FUNCTION_BLOCK FB_Snake EXTENDS FB_Glowny
VAR

	poleGry:S_Macierz;	
	
	wiersz:INT;//potem usunąć oba
	kolumna:INT;
	
	stanGry:INT:=3;

	iLicznikPrendkosci: INT;

	
	GAMEOVER:BOOL:=TRUE;
	EKRANSTARTOWY:BOOL:=FALSE;
	
	kierunek: INT;
	iLicznikKierunku: INT;
	kierunekRuchu:E_kierunek;
	
	stanJedzenia:BOOL;
	jedzeniePozycjaX:INT;
	jedzeniePozycjaY:INT;
	
	iLicnikPunktow:INT:=1;
	
	iWektorOgonaX:ARRAY[2..400] OF INT;
	iWektorOgonaY:ARRAY[2..400] OF INT;
	iLicznikY:INT:=2;

END_VAR

CASE stanGry OF
	
0:	
	FOR iLicznikKierunku:=1 TO 4  DO
		IF GVL_Lista.bStanStrzalek[iLicznikKierunku]=TRUE THEN
			kierunek:=iLicznikKierunku;							//sprawdzanie obecnego kierunku ruchu
			IF kierunek=1 THEN
				kierunekRuchu:=1;
			END_IF
			IF kierunek=2 THEN
				kierunekRuchu:=2;
			END_IF
			IF kierunek=3 THEN
				kierunekRuchu:=3;
			END_IF
			IF kierunek=4 THEN
				kierunekRuchu:=4;
			END_IF
		END_IF
	END_FOR
	M_SprawdzanieKolizji();
	IF stanJedzenia=FALSE THEN									//jeśli zdobędziemy punkt generuje nowe do zdobycia
		M_GenerowanieJedzenia();
	END_IF
	
	SUPER^.timerRuchu(IN:=TRUE,PT:=INT_TO_TIME(1000-(iLicznikPrendkosci*iLicnikPunktow))); //czas pomiędzy kolejnymi rychami 
	IF timerRuchu.Q=TRUE THEN
		IF  kierunek=1 THEN						//lewo
			iLicznikY:=iLicznikY+1;
			iWektorOgonaX[iLicznikY]:=wiersz;
			iWektorOgonaY[iLicznikY]:=kolumna;
			wiersz:=wiersz-1;
		END_IF
		
		IF  kierunek=2 THEN						//dół
			iLicznikY:=iLicznikY+1;
			iWektorOgonaX[iLicznikY]:=wiersz;
			iWektorOgonaY[iLicznikY]:=kolumna;
			kolumna:=kolumna+1;
			
		END_IF
		
		IF  kierunek=3 THEN						//prawo
			iLicznikY:=iLicznikY+1;
			iWektorOgonaX[iLicznikY]:=wiersz;
			iWektorOgonaY[iLicznikY]:=kolumna;
			wiersz:=wiersz+1;
			
		END_IF
		
		IF  kierunek=4 THEN						//góra
			iLicznikY:=iLicznikY+1;
			iWektorOgonaX[iLicznikY]:=wiersz;
			iWektorOgonaY[iLicznikY]:=kolumna;
			kolumna:=kolumna-1;
			
		END_IF
		
		stanGry:=1;
		
		IF kolumna>10 OR wiersz>10 OR kolumna<1 OR wiersz<1 THEN	// detekcja kolizji z ścianą
		stanGry:=2;
		END_IF
	END_IF

1:
	poleGry.MacierzPola[kolumna][wiersz]:=TRUE;
	timerRuchu(IN:=FALSE);
	M_Ogon();
	
	IF timerRuchu.Q=FALSE THEN
		IF iLicznikPrendkosci<100 THEN
			iLicznikPrendkosci:=iLicznikPrendkosci+1;
		END_IF
		IF jedzeniePozycjaX=wiersz AND jedzeniePozycjaY=kolumna THEN
			stanJedzenia:=FALSE;
			iLicnikPunktow:=iLicnikPunktow+1;
		END_IF
		stanGry:=0;
	END_IF
	
	
2:	
	M_NowaGra();

3:
	IF GVL_Lista.bStanPRzyciskuStartu=TRUE THEN
		M_Start();
	END_IF
END_CASE

METHOD M_GenerowanieJedzenia : BOOL
VAR
	iLicznik:INT;
END_VAR

jedzeniePozycjaX:=((iLicznikPrendkosci+wiersz) MOD 10)+1;	// z powodu iż w Twincacie nie mogłem znaleść funkcji RANDOM napisałem coś tkaiego, działa ale jest mało losowe
IF jedzeniePozycjaX <5 THEN
	jedzeniePozycjaX:=jedzeniePozycjaX + 2;
END_IF
jedzeniePozycjaY:=((jedzeniePozycjaX+kolumna) MOD 10)+1;
IF jedzeniePozycjaY<5 THEN
	jedzeniePozycjaY:=((jedzeniePozycjaY+wiersz) MOD 10)+1;
END_IF
IF jedzeniePozycjaX =wiersz OR jedzeniePozycjaY = kolumna THEN
	jedzeniePozycjaX:=((jedzeniePozycjaX+8) MOD 10)+1;
	jedzeniePozycjaY:=((jedzeniePozycjaX*jedzeniePozycjaY*iLicznikPrendkosci) MOD 10)+1; 
END_IF
poleGry.MacierzPola[jedzeniePozycjaY][jedzeniePozycjaX]:=TRUE;
StanJedzenia:=TRUE;
END_METHOD

METHOD M_NowaGra : BOOL
VAR
	i: INT;
	x: INT;
END_VAR
	poleGry.MacierzPola[jedzeniePozycjaY][jedzeniePozycjaX]:=FALSE;	
	GAMEOVER:=FALSE;													//wyłączenie informacji o przegranej grze
	IF iLicnikPunktow>GVL_Lista.iRekord THEN
		GVL_Lista.iRekord:=iLicnikPunktow;								// zapisanie liczby uzyskanych punktów
	END_IF
	FOR i:=1 TO 10 DO
		FOR x:=1 TO 10 DO
			poleGry.MacierzPola[x][i]:=FALSE;							// wyłączenie wszystkich pól
		END_FOR
	END_FOR
	IF GVL_Lista.bStanPrzyciskuRestart=TRUE THEN						//To samo co w przypadku metody M_Start
		THIS^.kolumna:=5;
		THIS^.wiersz:=6;
		THIS^.iWektorOgonaX[2]:=kolumna;
		THIS^.iWektorOgonaY[2]:=wiersz;
		THIS^.iLicznikY:=2;
		THIS^.kierunek:=0;
		THIS^.iLicnikPunktow:=1;
		THIS^.GAMEOVER:=TRUE;
		THIS^.iLicznikPrendkosci:=1;
		THIS^.stanJedzenia:=FALSE;
		THIS^.stanGry:=0;
	END_IF
END_METHOD

METHOD M_Ogon : BOOL
VAR
	//petla 1
	i:INT;
	x:INT;
	licznikOgona:INT;
	
	//liczenie co co skasowac
	q:INT;
	w:INT;
	
END_VAR
FOR i:=1 TO 10 DO
	FOR x:=1 TO 10 DO
		IF poleGry.MacierzPola[x][i]=TRUE THEN			
			licznikOgona:=licznikOgona+1;				//Pętal sprawdzająca czy długość = liczba punktów kiedy zdobędziemy punkt zwieksza długość
		END_IF
	END_FOR
END_FOR

IF (licznikOgona-1)>=iLicnikPunktow THEN
	q:=iWektorOgonaY[iLicznikY-(iLicnikPunktow-1)];	
	w:=iWektorOgonaX[iLicznikY-(iLicnikPunktow-1)];
	poleGry.MacierzPola[q][w]:=FALSE;					//usuwanie końca ogona
END_IF
END_METHOD

METHOD M_SprawdzanieKolizji : BOOL
VAR
	
	x:INT;
	
END_VAR
FOR x:=(iLicznikY-(iLicnikPunktow-1)) TO iLicznikY DO
	IF kierunek>0 THEN
			IF iWektorOgonaY[x]=kolumna AND iWektorOgonaX[x]=wiersz THEN	//jeżeli obecny stan kolumny i wierszu jest równy stanowi poprzedniemu -n to...
				stanGry:=2;													//to zmień stan gry
			END_IF
	END_IF
END_FOR
END_METHOD

METHOD M_Start : BOOL
VAR_INPUT
END_VAR
										//parametry zmiennych potrzebe przy starcie
	THIS^.kolumna:=6;  					//kolumna startowa
	THIS^.wiersz:=5;					//wiersz startowy
	THIS^.iWektorOgonaX[2]:=kolumna;	//macierz zapamiętujaca poprzednie stany
	THIS^.iWektorOgonaY[2]:=wiersz;
	THIS^.iLicznikPrendkosci:=1;		//restart prędkości
	THIS^.stanJedzenia:=FALSE;			//zmienna uruchamiająca proces tworzenia 'jedzenia dla wężyka'
	THIS^.EKRANSTARTOWY:=TRUE;			//wyłaczenie komunikatu
	THIS^.stanGry:=0;					//zmeina stanu programu
END_METHOD

END_FUNCTION_BLOCK

(* stored: Version 1.1.0.1, ProductVersion 3.1.4024.4
   POU FB_Snake: Id {31d2fabe-7c50-423b-aa7d-c8ea19a5f486}, SpecialFunc None
   Method M_GenerowanieJedzenia: Id {c227e4b4-9052-4591-9ec6-42f23383027a}
   Method M_NowaGra: Id {ab4a8c2d-5e84-4607-b7a3-15dfdf1bccdd}
   Method M_Ogon: Id {ea3cc6af-7f3a-474d-a684-7da53207cf11}
   Method M_SprawdzanieKolizji: Id {9e87a71a-75a5-459c-b349-562cf7ce5c7a}
   Method M_Start: Id {0c866838-f915-49db-ab4d-a12a741af533} *)
